INTERFACE I_ListOfInterfaces EXTENDS I_ListItem

METHOD AddInterface
VAR_INPUT
    InterfacePointer : I_ListItem;
END_VAR
END_METHOD

PROPERTY Count : DINT
GET
END_GET
END_PROPERTY

METHOD GetInterface : I_ListItem
VAR_INPUT
    Index : DINT;
END_VAR
END_METHOD

END_INTERFACE

(* stored: Version 1.1.0.1, ProductVersion 3.1.4024.12
   Itf I_ListOfInterfaces: Id {893e7e43-a7a7-456e-9517-e3d21b74d5fa}
   Method AddInterface: Id {e9ad3765-0af3-47ea-a604-b236c0477164}
   Property Count: Id {cd9ef367-f066-49ff-883b-2dba33c01866}
   Get Get: Id {b7f24ab7-3fd8-4494-9397-81af06512e9e}
   Method GetInterface: Id {bc5e0acc-0aa8-4117-b203-55864887c248} *)
